INTERFACE ITF_SITP_PolecenieZmianyTrybu EXTENDS ITF_SITP_PolecenieZmiany

METHOD PUBLIC zwrocRodzajPolecenia : E_SITP_PolecenieZmianyTrybu
VAR_INPUT
END_VAR
END_METHOD

END_INTERFACE

(* stored: Version 1.1.0.1
   Itf ITF_SITP_PolecenieZmianyTrybu: Id {e6d365c8-3885-057a-158d-3555cf440771}
   Method zwrocRodzajPolecenia: Id {832458fa-c954-0034-032b-ceefb46e3b2b} *)
